// TIA Portal project "HW_Plc1518V3_IndraDrive" (V18)

(* hardware
DEVICE "S71500/ET200MP station_2"  S7-1500 station
   slot 0: "Rail_0"  Rack  6ES7 590-1***0-0AA0
   slot 1: "PLC_LINE"  CPU 1518F-4 PN/DP  6ES7 518-4FP00-0AB0  V3.0
      slot 3: "CPU display_1"  6ES7591-1BA00-0AA0
      slot 32768: "PROFINET interface_1"  X1
      slot 33024: "PROFINET interface_2"  X2
      slot 33280: "PROFINET interface GBIT_3"  X3
      slot 33536: "DP interface_1"  X4
      slot 34817: "Virtual CP interface port_1"  Virtual CP interface port  Virtual CP interface port
DEVICE "CVIC II R2 A"  GSD.Device.PN
   slot 0: "Rack"  Rail  V1.0
   slot 0: "wp462-t1-rh-deso"  ABCC-PRT  V1.11
   slot 1: "Input 1 byte_1"  ABCC-PRT  V1.0
   slot 2: "Input 1 byte_2"  ABCC-PRT  V1.0
   slot 3: "Input 2 word_1"  ABCC-PRT  V1.0
   slot 4: "Input 1 word_1"  ABCC-PRT  V1.0
   slot 5: "Input 2 word_2"  ABCC-PRT  V1.0
   slot 6: "Input 1 word_2"  ABCC-PRT  V1.0
   slot 7: "Output 1 byte_1"  ABCC-PRT  V1.0
   slot 8: "Output 1 byte_2"  ABCC-PRT  V1.0
*)

// ===== PLC "PLC_LINE"  CPU 1518F-4 PN/DP =====

ORGANIZATION_BLOCK "Main"   // OB1, SCL, ProgramCycle
TITLE = "Main Program Sweep (Cycle)"
{ S7_Optimized_Access := 'FALSE' }
VERSION : 0.1
   VAR_TEMP
      EV_CLASS : Byte;   // Bits 0-3 = 1:Coming event, Bits 4-7 = 1:Event class 1
      SCAN_1 : Byte;   // 1:Initial call of the OB, 3: Call 2-n of the OB
      PRIORITY : Byte;   // Priority of OB Execution
      OB_NUMBR : Byte;   // OB number
      RESERVED_1 : Byte;   // Reserved for system
      RESERVED_2 : Byte;   // Reserved for system
      PREV_CYCLE : Int;   // Previous program cycle time (milliseconds)
      MIN_CYCLE : Int;   // Minimum program cycle time (milliseconds)
      MAX_CYCLE : Int;   // Maximum program cycle time (milliseconds)
      DATE_TIME : Date_And_Time;   // Date and time OB started
      SYSTEM_TIME : DTL;
      LOCAL_TIME : DTL;
   END_VAR
BEGIN
END_ORGANIZATION_BLOCK